{attribute 'qualified_only'}
{attribute 'strict'}
TYPE eErrorClearWays :
(
	NO_ACTION:=0,
	RESET := 1,
	IGNORE :=2
);
END_TYPE

(* stored: Version 1.1.0.1, ProductVersion 3.1.4022.10
   DUT eErrorClearWays: Id {541fffb7-8b44-45bb-b200-d22fefd5ea0c} *)
